FUNCTION_BLOCK fb_ConnectDB
VAR_INPUT
	DBInfo:st_DBInfo;
	bConnect:BOOL:=FALSE;
	
END_VAR
VAR_OUTPUT
	bConnected:BOOL:=FALSE;
END_VAR
VAR
END_VAR

METHOD connect : BOOL
VAR_INPUT
END_VAR
bConnect:=true;
END_METHOD

METHOD disconnect : BOOL
VAR_INPUT
END_VAR
bConnect:=false;
END_METHOD

END_FUNCTION_BLOCK

(* stored: Version 1.1.0.1, ProductVersion 3.1.4024.2
   POU fb_ConnectDB: Id {73f5ef1b-7b68-4a01-990c-094b461c6649}, SpecialFunc None
   Method connect: Id {3a3b9865-b3bf-4add-99b3-5aef312ac18a}
   Method disconnect: Id {b4bcc148-299b-4c24-93db-7a704b438317} *)
